// TIA Portal project "在PID学习中" (V16)

(* hardware
DEVICE "S71500/ET200MP station_2"  S7-1500 station
   slot 0: "导轨_0"  Rack  6ES7 590-1***0-0AA0
   slot 1: "PLC_2"  CPU 1511-1 PN  6ES7 511-1AK02-0AB0  V2.8
      slot 3: "CPU 显示_1"  6ES7591-1AA00-0AA0
      slot 32768: "PROFINET 接口_1"  X1
         slot 32769: "端口_1"  X1 P1
         slot 32770: "端口_2"  X1 P2
      slot 34817: "Virtual CP interface port_1"  Virtual CP interface port  Virtual CP interface port
DEVICE "S71500/ET200MP station_1"  S7-1500 station
   slot 0: "导轨_0"  Rack  6ES7 590-1***0-0AA0
   slot 1: "PLC_1"  CPU 1511C-1 PN  6ES7 511-1CK01-0AB0  V2.8
      slot 3: "CPU 显示_1"  6ES7591-1AA00-0AA0
      slot 32768: "PROFINET 接口_1"  X1
         slot 32769: "端口_1"  X1 P1
         slot 32770: "端口_2"  X1 P2
      slot 34817: "Virtual CP interface port_1"  Virtual CP interface port  Virtual CP interface port
*)

// ===== PLC "PLC_2"  CPU 1511-1 PN =====

VAR_GLOBAL   // PLC tag table "变量表_1"
   "启动开关" AT %I2.0 : Bool;
   "复位开关" AT %I2.1 : Bool;
   "停止开关" AT %I2.2 : Bool;
   "FACTORY I/O (Running)" AT %I2.3 : Bool;
   "启动指示灯" AT %Q2.0 : Bool;
   "复位指示灯" AT %Q2.1 : Bool;
   "停止指示灯" AT %Q2.2 : Bool;
   "液位计" AT %ID30 : Real;
   "流量计" AT %ID34 : Real;
   "定位点" AT %ID38 : Real;
   "进水阀" AT %QD30 : Real;
   "排出阀" AT %QD34 : Real;
   "流液显示屏" AT %QD38 : DInt;
   "流量显示屏" AT %QD42 : DInt;
END_VAR

DATA_BLOCK "数据块_1"   // DB1
{ S7_Optimized_Access := 'TRUE' }
VERSION : 0.1
   VAR
      设定值 : Real;
      输出值 : Real;
      报警 : DWord;
      解警 : Bool;
      转换值1 : Real;
      转换值2 : Real;
      实际值 : Real;
   END_VAR
BEGIN
END_DATA_BLOCK

ORGANIZATION_BLOCK "Main"   // OB1, LAD, ProgramCycle
TITLE = "Main Program Sweep (Cycle)"
{ S7_Optimized_Access := 'TRUE' }
VERSION : 0.1
   VAR_INPUT
      Initial_Call : Bool;   // Initial call of this OB
      Remanence : Bool;   // =True, if remanent data are available
   END_VAR
BEGIN

REGION Network 2
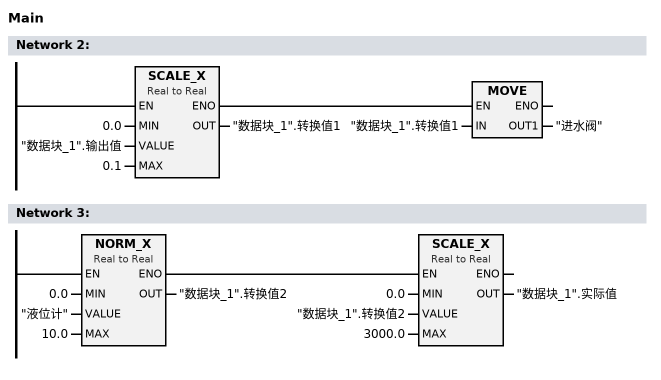
   RUNG wire#powerrail
      { S7_Templates := "[SrcType := Real, DestType := Real]" } Scale(min := 0.0, value := "数据块_1".输出值, max := 0.1, out => "数据块_1".转换值1)
      Move(in := "数据块_1".转换值1, out1 => "进水阀")
   END_RUNG
   // the same network as SCL:
   "数据块_1".转换值1 := SCALE_X(MIN := 0.0, VALUE := "数据块_1".输出值, MAX := 0.1);
   "进水阀" := "数据块_1".转换值1;
END_REGION

REGION Network 3
   RUNG wire#powerrail
      { S7_Templates := "[SrcType := Real, DestType := Real]" } Normalize(min := 0.0, value := "液位计", max := 10.0, out => "数据块_1".转换值2)
      { S7_Templates := "[SrcType := Real, DestType := Real]" } Scale(min := 0.0, value := "数据块_1".转换值2, max := 3000.0, out => "数据块_1".实际值)
   END_RUNG
   // the same network as SCL:
   "数据块_1".转换值2 := NORM_X(MIN := 0.0, VALUE := "液位计", MAX := 10.0);
   "数据块_1".实际值 := SCALE_X(MIN := 0.0, VALUE := "数据块_1".转换值2, MAX := 3000.0);
END_REGION
END_ORGANIZATION_BLOCK

ORGANIZATION_BLOCK "Cyclic interrupt"   // OB30, LAD, CyclicInterrupt
{ S7_Optimized_Access := 'TRUE' }
VERSION : 0.1
   VAR_INPUT
      Initial_Call : Bool;   // Initial call of this OB
      Event_Count : Int;   // Events discarded
   END_VAR
BEGIN

REGION Network 1
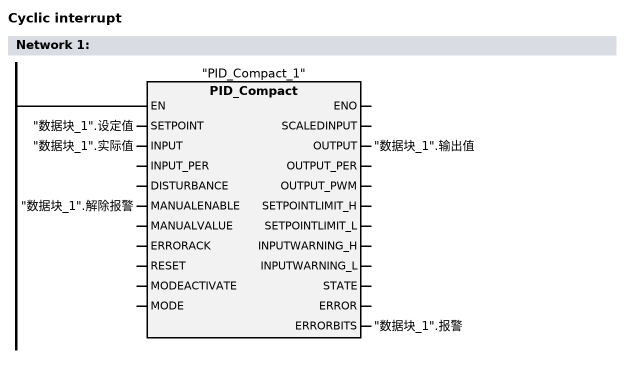
   "PID_Compact_1"(Setpoint := "数据块_1".设定值,   // PID_Compact
                   Input := "数据块_1".实际值,
                   ManualEnable := "数据块_1".解除报警,
                   Output => "数据块_1".输出值,
                   ErrorBits => "数据块_1".报警);
END_REGION
END_ORGANIZATION_BLOCK

// ===== PLC "PLC_1"  CPU 1511C-1 PN =====

ORGANIZATION_BLOCK "Main"   // OB1, LAD, ProgramCycle
TITLE = "Main Program Sweep (Cycle)"
{ S7_Optimized_Access := 'TRUE' }
VERSION : 0.1
   VAR_INPUT
      Initial_Call : Bool;   // Initial call of this OB
      Remanence : Bool;   // =True, if remanent data are available
   END_VAR
BEGIN
END_ORGANIZATION_BLOCK